# EPICS StreamDevice protocol: protocols/acq400mb.proto
Terminator = LF;
ExtraInput = Ignore;

# dma_stat_desc_push
# reply: count flags
# 62 0

# fails .. descr too long..
getFifo {
	out "\$1";
	in "%d %(\$2)d";
}

getFifoStatus {
	out "\$1";
	in "%*d %d";
}

getAggregator {
	out "aggregator";
	in "reg=0x%x sites=%*s threshold=%*d DATA_MOVER_EN=%*s";
}

getAggregatorSites {
	in "reg=0x%*x sites=%s threshold=%*d DATA_MOVER_EN=%*s";
}
#acq1102_005> cat /var/log/run0.log
#/usr/local/bin/run0 2,1 1,3,1 ssb=64

getAggregatorS1 {
        out "run0_log";
	in "%*s %d";
}

getAggregatorBackpressure {
        out "aggsta_backpressure";
	in "%d";
}

getAggregatorEn {
	in "reg=0x%*x sites=%*s threshold=%*d DATA_MOVER_EN=%{off|on}";
}

getDistributor {
	out "distributor";
	in "reg=0x%08x sites=%*s comms=%*s";
};

getDistributorSites{
	in "reg=0x%*08x sites=%s comms=%*s";
}

getDistributorS1{
	in "reg=0x%*08x sites=%d%*s comms=%*s";
}

getDistributorComms{
	in "reg=0x%*08x sites=%*s comms=%{9|B|A|U} pad=%*d";
}

getDistributorPad{
	in "reg=0x%*08x sites=%*s comms=%*s pad=%d";
}

getDistributorEn {
	in "reg=0x%*08x sites=%*s comms=%*s pad=%*d DATA_MOVER_EN=%{off|on}";
}

setDistributorSites {
	out "distributor sites=%s";
	in;
}

getHasMgt {
	out "has_mgt";
	in "%10c";
}

getString {
	out "\$1";
	in "%10c";
}

setStreamSubsetMask {
        out "stream_subset_mask %s";
        in;
}

getStreamSubsetMask {
        out "stream_subset_mask";
        in "%s";
}
